// ---- Visualizations/Pallettizzatore.TcVIS
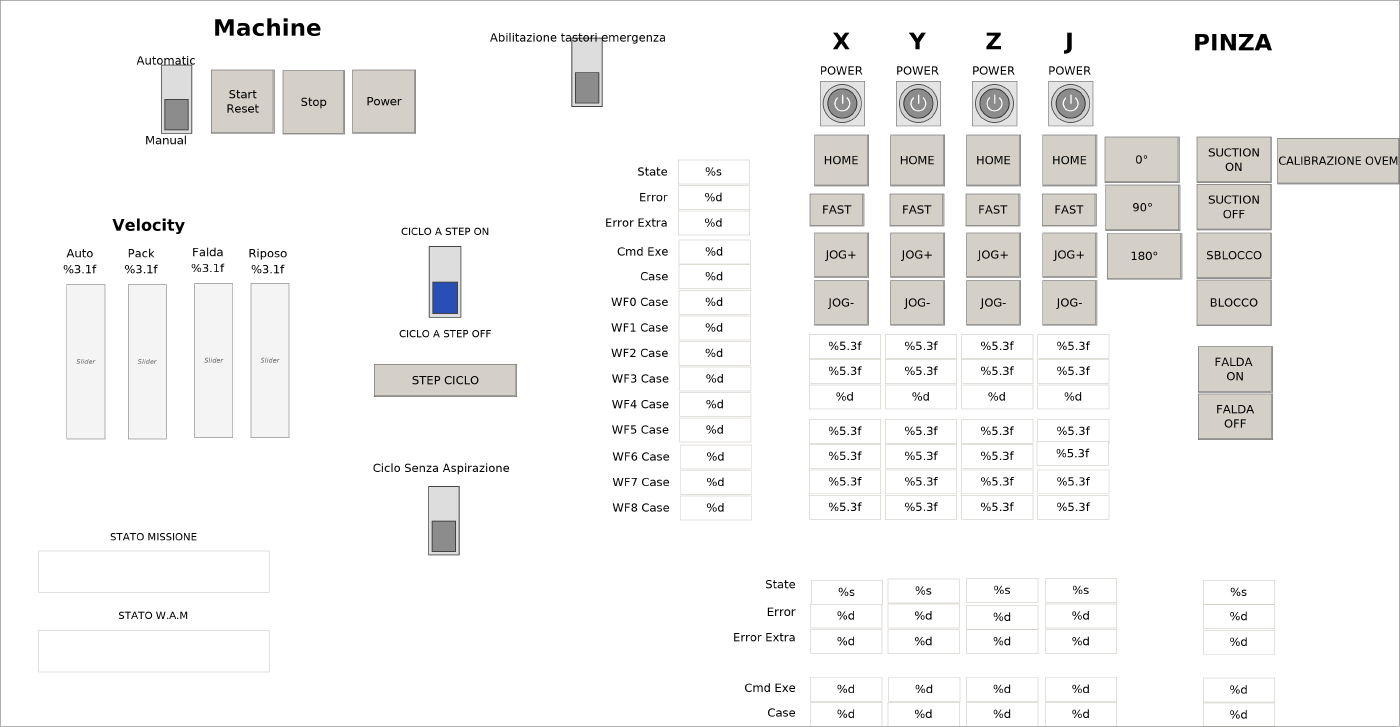
VISUALIZATION Pallettizzatore  // 2189x1138
    Label (295,15 246x57), "Machine"
    Label (213,205 94x30), "Manual"
    DipSwitch (209,101 134x108), variable: I_AutoPal, behaviour: TOGGLE, style: Switch-DipSwitch-Gray
    Label (213,80 94x30), "Automatic"
    Button (442,110 97x100), "Stop"
        tap HMI_Stop
    Button (330,109 99x100), "Start Reset"
        tap I_StartCicloPal
    Label (188,332 94x54)
    PowerSwitch (1282,127 70x70), variable: X_AxisLib.Command.Power, behaviour: TOGGLE, style: Switch-PowerSwitch-Gray
    Label (1287,36 57x57), "X"
    Label (1272,96 87x30), "POWER"
    Button (1273,364 85x70), "JOG+"
        tap MachinePalletizer_TF.ManCmd^.X.JogPos
    Button (1273,439 85x70), "JOG-"
        tap MachinePalletizer_TF.ManCmd^.X.JogNeg
    Button (1273,211 85x80), "HOME"
        OnMouseUp: execute { MachinePalletizer_TF.ManCmd^.X.Home := TRUE; }
    Button (1266,303 85x51), "FAST", colour toggle: MachinePalletizer_TF.ManCmd^.X.JogFast
        toggle MachinePalletizer_TF.ManCmd^.X.JogFast p2164770859=TRUE
    PowerSwitch (1401,127 70x70), variable: Y_AxisLib.Command.Power, behaviour: TOGGLE, style: Switch-PowerSwitch-Gray
    Label (1406,36 57x57), "Y"
    Label (1391,96 87x30), "POWER"
    Button (1392,364 85x70), "JOG+"
        tap MachinePalletizer_TF.ManCmd^.Y.JogPos
    Button (1392,439 85x70), "JOG-"
        tap MachinePalletizer_TF.ManCmd^.Y.JogNeg
    Button (1392,211 85x80), "HOME"
        OnMouseUp: execute { MachinePalletizer_TF.ManCmd^.Y.Home := TRUE; }
    Button (1391,303 85x51), "FAST", colour toggle: MachinePalletizer_TF.ManCmd^.Y.JogFast
        toggle MachinePalletizer_TF.ManCmd^.Y.JogFast p2164770859=TRUE
    PowerSwitch (1520,127 70x70), variable: Z_AxisLib.Command.Power, behaviour: TOGGLE, style: Switch-PowerSwitch-Gray
    Label (1525,36 57x57), "Z"
    Label (1510,96 87x30), "POWER"
    Button (1511,364 85x70), "JOG+"
        tap MachinePalletizer_TF.ManCmd^.Z.JogPos
    Button (1511,439 85x70), "JOG-"
        tap MachinePalletizer_TF.ManCmd^.Z.JogNeg
    Button (1511,211 85x80), "HOME"
        OnMouseUp: execute { MachinePalletizer_TF.ManCmd^.Z.Home := TRUE; }
    Button (1510,303 85x51), "FAST", colour toggle: MachinePalletizer_TF.ManCmd^.Z.JogFast
        toggle MachinePalletizer_TF.ManCmd^.Z.JogFast
    PowerSwitch (1639,127 70x70), variable: J_AxisLib.Command.Power, behaviour: TOGGLE, style: Switch-PowerSwitch-Gray
    Label (1644,36 57x57), "J"
    Label (1629,96 87x30), "POWER"
    Button (1630,364 85x70), "JOG+"
        tap MachinePalletizer_TF.ManCmd^.J.JogPos
    Button (1630,439 85x70), "JOG-"
        tap MachinePalletizer_TF.ManCmd^.J.JogNeg
    Button (1630,211 85x80), "HOME"
        OnMouseUp: execute { MachinePalletizer_TF.ManCmd^.J.Home := TRUE; }
    Button (1629,303 85x51), "FAST", colour toggle: MachinePalletizer.ManCmd^.J.JogFast
        toggle MachinePalletizer_TF.ManCmd^.J.JogFast
    Textfield (1265,523 112x38), "%5.3f", text variable: X_AxisLib.Status.ActPosition
    Textfield (1265,562 112x38), "%5.3f", text variable: X_AxisLib.Status.ActVelocity
    Textfield (1265,656 112x38), "%5.3f", text variable: X_AxisLib.Parameter.Position
    Textfield (1265,695 112x38), "%5.3f", text variable: X_AxisLib.Parameter.Velocity
    Textfield (1265,735 112x38), "%5.3f", text variable: X_AxisLib.Parameter.Acceleration
    Textfield (1265,775 112x38), "%5.3f", text variable: X_AxisLib.Parameter.Deceleration
    Textfield (1384,523 112x38), "%5.3f", text variable: Y_AxisLib.Status.ActPosition
    Textfield (1384,562 112x38), "%5.3f", text variable: Y_AxisLib.Status.ActVelocity
    Textfield (1384,656 112x38), "%5.3f", text variable: Y_AxisLib.Parameter.Position
    Textfield (1384,695 112x38), "%5.3f", text variable: Y_AxisLib.Parameter.Velocity
    Textfield (1384,735 112x38), "%5.3f", text variable: Y_AxisLib.Parameter.Acceleration
    Textfield (1384,775 112x38), "%5.3f", text variable: Y_AxisLib.Parameter.Deceleration
    Textfield (1503,523 112x38), "%5.3f", text variable: Z_AxisLib.Status.ActPosition
    Textfield (1503,562 112x38), "%5.3f", text variable: Z_AxisLib.Status.ActVelocity
    Textfield (1503,656 112x38), "%5.3f", text variable: Z_AxisLib.Parameter.Position
    Textfield (1503,695 112x38), "%5.3f", text variable: Z_AxisLib.Parameter.Velocity
    Textfield (1503,735 112x38), "%5.3f", text variable: Z_AxisLib.Parameter.Acceleration
    Textfield (1503,775 112x38), "%5.3f", text variable: Z_AxisLib.Parameter.Deceleration
    Textfield (1622,523 112x38), "%5.3f", text variable: J_AxisLib.Status.ActPosition
    Textfield (1622,562 112x38), "%5.3f", text variable: J_AxisLib.Status.ActVelocity
    Textfield (1622,656 112x38), "%5.3f", text variable: J_AxisLib.Parameter.Position
    Textfield (1621,691 112x38), "%5.3f", text variable: J_AxisLib.Parameter.Velocity
    Textfield (1622,735 112x38), "%5.3f", text variable: J_AxisLib.Parameter.Acceleration
    Textfield (1622,775 112x38), "%5.3f", text variable: J_AxisLib.Parameter.Deceleration
    Textfield (1265,602 112x38), "%d", text variable: X_AxisLib.Status.ErrorID
    Textfield (1384,602 112x38), "%d", text variable: Y_AxisLib.Status.ErrorID
    Textfield (1503,602 112x38), "%d", text variable: Z_AxisLib.Status.ErrorID
    Textfield (1622,602 112x38), "%d", text variable: J_AxisLib.Status.ErrorID
    Textfield (1267,945 112x38), "%d", text variable: MachinePalletizerModules.AX_X.Error.Code
    Textfield (1268,908 112x38), "%s", text variable: MachinePalletizerModules.AX_X.State.Code
    Textfield (1267,1060 112x38), "%d", text variable: MachinePalletizerModules.AX_X.CmdExe.Code
    Textfield (1267,1099 112x38), "%d", text variable: MachinePalletizerModules.AX_X.CmdExe.CmdCase
    Textfield (1267,985 112x38), "%d", text variable: MachinePalletizerModules.AX_X.Error.ExtraCode
    Textfield (1388,945 112x38), "%d", text variable: MachinePalletizerModules.AX_Y.Error.Code
    Textfield (1388,906 112x38), "%s", text variable: MachinePalletizerModules.AX_Y.State.Code
    Textfield (1389,1060 112x38), "%d", text variable: MachinePalletizerModules.AX_Y.CmdExe.Code
    Textfield (1388,1099 112x38), "%d", text variable: MachinePalletizerModules.AX_Y.CmdExe.CmdCase
    Textfield (1388,985 112x38), "%d", text variable: MachinePalletizerModules.AX_Y.Error.ExtraCode
    Textfield (1511,947 112x38), "%d", text variable: MachinePalletizerModules.AX_Z.Error.Code
    Textfield (1511,905 112x38), "%s", text variable: MachinePalletizerModules.AX_Z.State.Code
    Textfield (1511,1060 112x38), "%d", text variable: MachinePalletizerModules.AX_Z.CmdExe.Code
    Textfield (1511,1099 112x38), "%d", text variable: MachinePalletizerModules.AX_Z.CmdExe.CmdCase
    Textfield (1511,985 112x38), "%d", text variable: MachinePalletizerModules.AX_Z.Error.ExtraCode
    Textfield (1634,945 112x38), "%d", text variable: MachinePalletizerModules.AX_J.Error.Code
    Textfield (1634,905 112x38), "%s", text variable: MachinePalletizerModules.AX_J.State.Code
    Textfield (1634,1060 112x38), "%d", text variable: MachinePalletizerModules.AX_J.CmdExe.Code
    Textfield (1634,1099 112x38), "%d", text variable: MachinePalletizerModules.AX_J.CmdExe.CmdCase
    Textfield (1634,985 112x38), "%d", text variable: MachinePalletizerModules.AX_J.Error.ExtraCode
    Textfield (1881,946 112x38), "%d", text variable: MachinePalletizerModules.Pinza.Error.Code
    Textfield (1881,908 112x38), "%s", text variable: MachinePalletizerModules.Pinza.State.Code
    Textfield (1881,1061 112x38), "%d", text variable: MachinePalletizerModules.Pinza.CmdExe.Code
    Textfield (1881,1100 112x38), "%d", text variable: MachinePalletizerModules.Pinza.CmdExe.CmdCase
    Textfield (1881,986 112x38), "%d", text variable: MachinePalletizerModules.Pinza.Error.ExtraCode
    Textfield (1060,290 112x38), "%d", text variable: MachinePalletizer_TF.Error.Code
    Textfield (1060,250 112x38), "%s", text variable: MachinePalletizer_TF.State.Code
    Textfield (1061,375 112x38), "%d", text variable: MachinePalletizer_TF.CmdExe.Code
    Textfield (1061,414 112x38), "%d", text variable: MachinePalletizer_TF.CmdExe.CmdCase
    Textfield (1061,454 112x38), "%d", text variable: MachinePalletizer_TF.WorkFlow[0].WFCase
    Textfield (1061,494 112x38), "%d", text variable: MachinePalletizer_TF.WorkFlow[1].WFCase
    Label (981,254 66x30), "State"
    Label (964,379 84x30), "Cmd Exe"
    Label (992,418 56x30), "Case"
    Label (956,458 92x30), "WF0 Case"
    Label (958,498 90x30), "WF1 Case"
    Label (991,294 56x30), "Error"
    Textfield (1061,534 112x38), "%d", text variable: MachinePalletizer_TF.WorkFlow[2].WFCase
    Label (958,538 90x30), "WF2 Case"
    Textfield (1060,330 112x38), "%d", text variable: MachinePalletizer_TF.Error.ExtraCode
    Label (943,334 104x30), "Error Extra"
    Textfield (1062,574 112x38), "%d", text variable: MachinePalletizer_TF.WorkFlow[3].WFCase
    Textfield (1062,614 112x38), "%d", text variable: MachinePalletizer_TF.WorkFlow[4].WFCase
    Label (957,578 92x30), "WF3 Case"
    Label (959,618 90x30), "WF4 Case"
    Textfield (1062,654 112x38), "%d", text variable: MachinePalletizer_TF.WorkFlow[5].WFCase
    Label (959,658 90x30), "WF5 Case"
    Textfield (1063,696 112x38), "%d", text variable: MachinePalletizer_TF.WorkFlow[6].WFCase
    Textfield (1063,736 112x38), "%d", text variable: MachinePalletizer_TF.WorkFlow[7].WFCase
    Label (958,700 92x30), "WF6 Case"
    Label (960,740 90x30), "WF7 Case"
    Textfield (1063,776 112x38), "%d", text variable: MachinePalletizer_TF.WorkFlow[8].WFCase
    Label (960,780 90x30), "WF8 Case"
    Button (551,109 99x100), "Power"
        tap I_PulsanteMarciaConsolle
    Label (1045,1062 202x30), "Cmd Exe"
    Label (1045,900 202x30), "State"
    Label (1045,1101 202x30), "Case"
    Label (1045,943 202x30), "Error"
    Label (1045,983 202x30), "Error Extra"
    Group (540,309 312x312)
        Button (45,261 223x51), "STEP CICLO", colour toggle: not MachinePalletizer.STEPCicloDONE
            tap HMI_CommandSTEP
        DipSwitch (100,73 112x118), variable: HMI_AbilitazioneCicloAStep, behaviour: TOGGLE, style: Switch-DipSwitch-Blue
        Label (0,0 312x107), "CICLO A STEP ON"
        Label (0,160 312x107), "CICLO A STEP OFF"
    Slider (104,445 60x242), variable: HMI_AxisOverride.Auto, scale 0..100
    Textfield (95,403 59x38), "%3.1f", text variable: HMI_AxisOverride.Auto
    Label (86,382 78x30), "Auto"
    Slider (200,445 60x242), variable: HMI_AxisOverride.Pack, scale 0..100
    Textfield (191,403 59x38), "%3.1f", text variable: HMI_AxisOverride.Pack
    Label (182,382 78x30), "Pack"
    Slider (392,443 60x242), variable: HMI_AxisOverride.PickRip, scale 0..100
    Textfield (389,403 59x38), "%3.1f", text variable: HMI_AxisOverride.PickRip
    Label (380,382 78x30), "Riposo"
    Label (129,337 207x30), "Velocity"
    Button (1871,214 117x72), "SUCTION ON"
        tap MachinePalletizer_TF.ManCmd^.Pinza.AttivazioneVuotoSX
    Button (1871,288 117x72), "SUCTION OFF"
        tap MachinePalletizer_TF.ManCmd^.Pinza.DisattivazioneVuotoSX
    Button (1871,364 117x72), "SBLOCCO"
        tap MachinePalletizer_TF.ManCmd^.Pinza.SbloccoPinza
    Button (1871,438 117x72), "BLOCCO"
        tap MachinePalletizer_TF.ManCmd^.Pinza.BloccoPinza
    Textfield (60,862 361x65), text list: 'Stato_Missione', text index: Mission.State
    Textfield (60,986 361x66), text list: 'Stato_WAM', text index: WorkAreaManager.State
    Label (84,787 312x107), "STATO MISSIONE"
    Label (84,910 312x107), "STATO W.A.M"
    DipSwitch (851,59 134x108), variable: TouchErrorEnable, behaviour: TOGGLE, style: Switch-DipSwitch-Gray
    Label (759,44 290x30), "Abilitazione tastori emergenza"
    DipSwitch (627,761 134x108), variable: HMI_AbilitaSimulazioneAVuoto, behaviour: TOGGLE, style: Switch-DipSwitch-Gray
    Label (545,718 290x30), "Ciclo Senza Aspirazione"
    Label (1859,38 137x57), "PINZA"
    Button (1873,542 117x72), "FALDA ON"
        tap MachinePalletizer_TF.ManCmd^.Pinza.AttivazioneVuotoFaldeSX
    Button (1873,616 117x72), "FALDA OFF"
        tap MachinePalletizer_TF.ManCmd^.Pinza.DisattivazioneVuotoFaldeSX
    Button (1727,214 117x72), "0°"
        tap MachinePalletizer_TF.ManCmd^.PosizionamentoPinza0
    Button (1728,289 117x72), "90°"
        tap MachinePalletizer_TF.ManCmd^.PosizionamentoPinza90
    Button (1731,365 117x72), "180°"
        tap MachinePalletizer_TF.ManCmd^.PosizionamentoPinza180
    Button (1997,216 192x72), "CALIBRAZIONE OVEM"
        tap MachinePalletizer_TF.ManCmd^.Pinza.CalibrazioneOVEM
    Label (286,380 78x30), "Falda"
    Slider (304,443 60x242), variable: HMI_AxisOverride.Layer, scale 0..100
    Textfield (295,401 59x38), "%3.1f", text variable: HMI_AxisOverride.Layer
END_VISUALIZATION

// ---- Visualizations/Stato_Missione.TcTLO
TEXTLIST Stato_Missione
  0 = 'NOP'
  999 = 'ERROR'
  30 = 'PRELIEVO PALLET RUN'
  31 = 'PRELIEVO PALLET END'
  40 = 'DEPOSITO PALLET RUN'
  41 = 'DEPOSITO PALLET END'
  20 = 'VAI A RIPOSO RUN'
  21 = 'VAI A RIPOSO END'
  50 = 'PRELIEVO FALDA RUN'
  51 = 'PRELIEVO FALDA END'
  60 = 'DEPOSITO FALDA RUN'
  61 = 'DEPOSITO FALDA END'
  70 = 'PRELIEVO PACCO RUN'
  71 = 'PRELIEVO PACCO END'
  80 = 'DEPOSITO PACCO RUN'
  81 = 'DEPOSITO PACCO END'
  10 = ''
  90 = 'PRELIEVO LASTRA RUN'
  91 = 'PRELIEVO LASTRA END'
  100 = 'DEPOSITO LASTRA RUN'
  101 = 'DEPOSITO LASTRA END'
   = ''
END_TEXTLIST

// ---- Visualizations/Stato_WAM.TcTLO
TEXTLIST Stato_WAM
  100 = 'IN ATTESA DI MISSIONE'
  111 = 'CICLO RIPOSO INIT'
  112 = 'CICLO RIPOSO RUN'
  113 = 'WAM CICLO RIPOSO END'
  120 = 'WAM CICLO PALLET INIT'
  121 = 'WAM CICLO PRELIEVO PALLET RUN'
  122 = 'WAM CICLO PRELIEVO PALLET END'
  123 = 'WAM CICLO DEPOSITO PALLET RUN'
  124 = 'WAM CICLO DEPOSITO PALLET END'
  130 = 'WAM CICLO FALDA VUOTI INIT'
  131 = 'WAM CICLO PRELIEVO FALDA VUOTI RUN'
  132 = 'WAM CICLO PRELIEVO FALDA VUOTI END'
  133 = 'WAM CICLO DEPOSITO FALDA VUOTI RUN'
  134 = 'WAM CICLO DEPOSITO FALDA VUOTI END'
  140 = 'WAM CICLO FALDA INIT'
  141 = 'WAM CICLO PRELIEVO FALDA RUN'
  142 = 'WAM CICLO PRELIEVO FALDA END'
  143 = 'WAM CICLO DEPOSITOFALDA RUN'
  144 = 'WAM CICLO DEPOSITO FALDA END'
  150 = 'WAM CICLO PACCO INIT'
  151 = 'WAM CICLO PRELIEVO PACCO RUN'
  152 = 'WAM CICLO PRELIEVO PACCO END'
  153 = 'WAM CICLO DEPOSITO PACCO RUN'
  154 = 'WAM CICLO DEPOSITO PACCO END'
  200 = 'WAMANAGER_CICLO_PRELIEVO_LASTRA_PANCONE_INIT'
  201 = 'CICLO PRELIEVO LASTRA DA PANCONE RUN\n'
  202 = 'WAMANAGER_CICLO_PRELIEVO_LASTRA_DA_PANCONE_END'
  203 = 'WAMANAGER_CICLO_DEPOSITO_LASTRA_PANCONE_INIT'
  204 = 'CICLO DEPOSITO LASTRA SU PANCONE RUN'
  205 = 'WAMANAGER_CICLO_DEPOSITO_LASTRA_SU_PANCONE_END'
  206 = 'WAMANAGER_CICLO_PRELIEVO_LASTRA_DA_CANTILEVER_INIT'
  207 = 'CICLO PRELIEVO LASTRA DA CANTILEVER RUN'
  208 = 'WAMANAGER_CICLO_PRELIEVO_LASTRA_DA_CANTILEVER_END'
  209 = 'WAMANAGER_CICLO_DEPOSITO_LASTRA_SU_CANTILEVER_INIT'
  210 = 'CICLO DEPOSITO LASTRA SU CANTILEVER RUN'
  211 = 'CICLO DEPOSITO LASTRA SU CANTILEVER END'
  212 = 'WAMANAGER_CICLO_POSIZIONAMENTO_SEMPLICE_INIT'
  213 = 'CICLO POSIZIONAMENTO SEMPLICE'
  214 = 'WAMANAGER_CICLO_POSIZONAMENTO_SEMPLICE_END'
  170 = 'WAM CICLO LASTRA INIT'
  171 = 'WAM CICLO PRELIEVO LASTRA RUN'
  172 = 'WAM CICLO PRELIEVO LASTRA END'
  173 = 'WAM CICLO DEPOSITO LASTRA RUN'
  174 = 'WAM CICLO DEPOSITO LASTRA END'
   = ''
END_TEXTLIST
